# EPICS StreamDevice protocol: piSerial/serialClient/proto/client.proto
Terminator = LF;
ReplyTimeout = 1000;

get_ai_data {
	out "\$1";
	in "%f";
}

get_bi_data {
	out "\$1";
	in "%d";
}
